PROGRAM Main
VAR
	CoreSwaging: FB_CoreSwaging;
    OilPump: FB_OilPump;
    CorePress: FB_CorePress;
    CasingVibratoryBowl1: FB_CasingVibratoryBowl1;
    CoreVibratoryBowl2: FB_CoreVibratoryBowl2;

	bCoreSwagingFaulted: BOOL := FALSE;
	bOilPumpFaulted: BOOL := FALSE;
	bCorePressFaulted: BOOL := FALSE;
	bCasingVibratoryBowl1Faulted: BOOL := FALSE;
	bCoreVibratoryBowl2Faulted: BOOL := FALSE;
    bAnyRoutineFaulted: BOOL := FALSE;
END_VAR

IF NOT bAnyRoutineFaulted THEN
	CoreSwaging(i_bEnabled := TRUE);
	OilPump(i_bEnabled := TRUE);
	CorePress(i_bEnabled := TRUE);
	CasingVibratoryBowl1(i_bEnabled := TRUE);
	CoreVibratoryBowl2(i_bEnabled := TRUE);
	
	bCoreSwagingFaulted := CoreSwaging.o_bFaulted;
	bOilPumpFaulted := OilPump.o_bFaulted;
	bCorePressFaulted := CorePress.o_bFaulted;
	bCasingVibratoryBowl1Faulted := CasingVibratoryBowl1.o_bFaulted;
	bCoreVibratoryBowl2Faulted := CoreVibratoryBowl2.o_bFaulted;
	bAnyRoutineFaulted := bCoreSwagingFaulted OR bOilPumpFaulted
							OR bCorePressFaulted OR bCasingVibratoryBowl1Faulted OR bCoreVibratoryBowl2Faulted;
END_IF

GVL_IO.DO_LGreen := NOT bAnyRoutineFaulted;
GVL_IO.DO_LRed := bAnyRoutineFaulted;

END_PROGRAM

(* stored: Version 1.1.0.1, ProductVersion 3.1.4024.6
   POU MAIN: Id {a9276fae-2b8f-4b86-a5ea-ccb7b5233763}, SpecialFunc None *)
